{attribute 'qualified_only'}
{attribute 'strict'}
TYPE E_Mechanische_Stop :
(
	enum_member := 0
);
END_TYPE

(* stored: Version 1.1.0.1, ProductVersion 3.1.4024.12
   DUT E_Mechanische_Stop: Id {2d24695f-828e-4a06-9de1-831f231ceaa6} *)
